FUNCTION_BLOCK FB_Window
VAR_INPUT
	Minimum:REAL;
	X:REAL;
	Maximum:REAL;
END_VAR
VAR_OUTPUT
	In_window:BOOL;
END_VAR
VAR
END_VAR

M_Window();

METHOD M_Window
VAR_INPUT
END_VAR
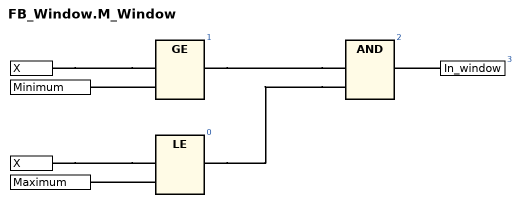
In_window := X >= Minimum AND X <= Maximum;
END_METHOD

END_FUNCTION_BLOCK

(* stored: Version 1.1.0.1, ProductVersion 3.1.4024.0
   POU FB_Window: Id {63b8565e-5435-4e4f-abdc-d4ff3128c167}, SpecialFunc None
   Method M_Window: Id {06f34b8d-b8c3-4b5f-b952-e2bf6be2e546} *)
